{attribute addProperty BoxType "EK1100-0000-0018"}
{attribute addProperty Id "Beckhoff_EPP9xxxEK1122Beckhoff_EPP9xxxEK1122_5167694C53266.5"}
{attribute addProperty CRC "2973246930"}
{attribute addProperty SizeInBites "532"}
{attribute addProperty SizeInBytes "66.5"}
TYPE Beckhoff_EPP9xxx_B13825D2 EXTENDS EK1100_179A0949 :
STRUCT
	{attribute addProperty Name "Beckhoff_EPP9xxxEK1122"}
	Beckhoff_EPP9xxxEK1122 : Beckhoff_EPP9xxxEK1122_5167694C;
END_STRUCT
END_TYPE

(* stored: Version 1.2.0.0, ProductVersion 3.1.4024.9
   DUT Beckhoff_EPP9xxx_B13825D2: Id {08e138ac-a925-411e-955a-f8eb5a26cb36} *)
